// TIA Portal V20 export
TYPE "typeFdoorCommands"
// stored: Access Published, IsFailsafeCompliant true, Namespace Safety
   STRUCT
      Lock : Bool;
      Unlock : Bool;
   END_STRUCT;
END_TYPE
